# EPICS substitutions: tests/example-config/ioc.substitutions
# Macros:
#  IOC  Device prefix
file $(IOCSTATS)/db/iocAdminSoft.db
{
pattern { IOC }
    { "test-ioc" }
}

# Macros:
#  IOC  Device prefix
file $(IOCSTATS)/db/iocAdminScanMon.db
{
pattern { IOC }
    { "test-ioc" }
}
